// TIA Portal V21 export
// export: Created 2026-07-12T08:36:11.2898125Z, ExportSetting None, DisplayName Totally Integrated Automation Portal, DisplayVersion V21, DisplayName SINAMICS Startdrive Advanced, DisplayVersion V21, DisplayName SINAMICS Startdrive G110M, G120, G120C, G120D, G120P, G115D, DisplayVersion V21, DisplayName SINAMICS Startdrive G130, G150, S120, S150, G200, G220, S200, S210, S220, Innomotics MVD, DisplayVersion V21, DisplayName STEP 7 Professional, DisplayVersion V21, DisplayName STEP 7 Safety, DisplayVersion V21, DisplayName Tech WebApplication, DisplayVersion V21, DisplayName WinCC Basic/Comfort/Advanced, DisplayVersion V21, DisplayName WinCC Professional, DisplayVersion V21, DisplayName WinCC Unified, DisplayVersion V21
FUNCTION_BLOCK "FB_SingleSolCyl_SCL"   // FB2104, LAD
{ S7_Optimized_Access := 'TRUE' }
// stored: AutoNumber false, MemoryReserve 100, SetENOAutomatically false
   VAR_INPUT
      Enable : Bool := 1;   // 使能单控气缸控制块，FALSE时关闭输出并禁止动作
      Mode : Int;   // 模式选择：1=Manual手动，2=Auto自动；其它值报警
      Exe_Auto : Bool;   // 自动模式下的动作命令，1伸出，0缩回
      Exe_Manual : Bool;   // 手动模式下的动作命令，1伸出，0缩回
      Sensor_Ext : Bool;   // 气缸伸出到位检测信号
      Sensor_Home : Bool;   // 气缸缩回原点检测信号
      Reset : Bool;   // 报警复位命令，清除报警和报警代码
      Timeout : Time := T#3S;   // 伸出或缩回等待传感器到位的超时时间，例如T#5s
   END_VAR
   VAR_OUTPUT
      Q : Bool;   // 控制真实电磁阀Q点，TRUE气缸伸出，FALSE气缸缩回
      Error : Bool;   // 报警锁存输出，需要ResetAlarm清除
      Error_Status : Word;   // 报警代码：2模式无效，3传感器冲突，257伸出超时，258缩回超时
      Extend : Bool;   // 当前有效模式下的伸出命令
      Retract : Bool;   // 当前有效模式下的缩回命令
      AutoActive : Bool;   // 自动模式有效状态：Enable、Mode=2、无报警
      ManualActive : Bool;   // 手动模式有效状态：Enable、Mode=1、无报警
   END_VAR
   VAR
      ExtendTimeoutTimer : TON_TIME;   // 伸出动作超时TON实例
      RetractTimeoutTimer : TON_TIME;   // 缩回动作超时TON实例
   END_VAR
BEGIN

REGION Network 1 (SCL): 条件判断集中处理
   // 报警、动作命令、伸出/缩回超时集中在本SCL程序段处理；ManualActive、AutoActive和Q输出保留LAD程序段。
   // 条件集中处理：报警、命令、超时都放在本SCL程序段
   // 保留LAD程序段只负责：ManualActive、AutoActive、Q输出

   // Reset优先清除报警；若故障原因仍存在，后续逻辑会重新报警
   IF #Reset THEN
       #Error := FALSE;
       #Error_Status := W#16#0000;
   END_IF;

   // 默认先清除动作命令，避免无效模式或报警时误动作
   #Extend := FALSE;
   #Retract := FALSE;

   // 根据有效模式生成动作命令：1伸出，0缩回
   IF #Enable AND NOT #Error THEN
       IF #ManualActive THEN
           #Extend := #Exe_Manual;
           #Retract := NOT #Exe_Manual;
       ELSIF #AutoActive THEN
           #Extend := #Exe_Auto;
           #Retract := NOT #Exe_Auto;
       END_IF;
   END_IF;

   // 定时器集中调用：伸出等待Sensor_Ext，缩回等待Sensor_Home
   #ExtendTimeoutTimer(IN := #Extend AND NOT #Sensor_Ext,
                       PT := #Timeout);
   #RetractTimeoutTimer(IN := #Retract AND NOT #Sensor_Home,
                        PT := #Timeout);

   // 报警判断集中处理
   IF #Enable AND NOT #Error THEN
       // Mode只能为1或2；
       IF (#Mode <> 1) AND (#Mode <> 2) THEN
           #Error := TRUE;
           #Error_Status := W#16#0002;

       // 两个极限传感器不能同时为1
       ELSIF #Sensor_Ext AND #Sensor_Home THEN
           #Error := TRUE;
           #Error_Status := W#16#0003;

       // 伸出不到位超时
       ELSIF #ExtendTimeoutTimer.Q THEN
           #Error := TRUE;
           #Error_Status := W#16#0101;

       // 缩回不到位超时
       ELSIF #RetractTimeoutTimer.Q THEN
           #Error := TRUE;
           #Error_Status := W#16#0102;
       END_IF;
   END_IF;

   // 报警后本扫描周期立即撤销有效模式和动作命令，后续LAD Q输出保持安全关闭
   IF #Error THEN
       #ManualActive := FALSE;
       #AutoActive := FALSE;
       #Extend := FALSE;
       #Retract := FALSE;
   END_IF;
END_REGION

REGION Network 2: Manual模式有效
   // Mode=1时手动模式有效，只允许ManualCmd控制气缸。
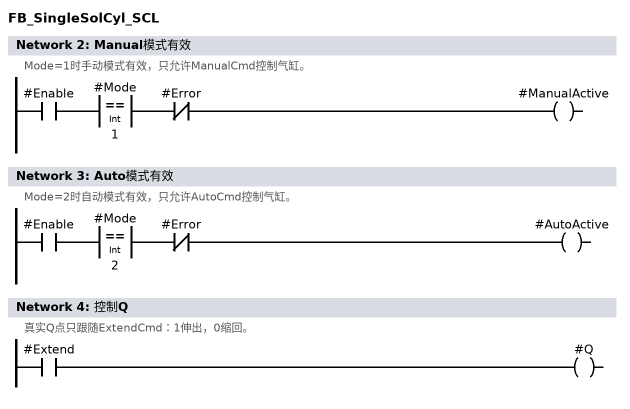
   RUNG wire#powerrail
      Contact( #Enable )
      { S7_Templates := "SrcType := Int" } EQ_Contact(in1 := #Mode, in2 := 1)
      I_Contact( #Error )
      Coil( #ManualActive )
   END_RUNG
   // the same network as SCL:
   #ManualActive := #Enable AND (#Mode = 1) AND NOT #Error;
END_REGION

REGION Network 3: Auto模式有效
   // Mode=2时自动模式有效，只允许AutoCmd控制气缸。
   RUNG wire#powerrail
      Contact( #Enable )
      { S7_Templates := "SrcType := Int" } EQ_Contact(in1 := #Mode, in2 := 2)
      I_Contact( #Error )
      Coil( #AutoActive )
   END_RUNG
   // the same network as SCL:
   #AutoActive := #Enable AND (#Mode = 2) AND NOT #Error;
END_REGION

REGION Network 4: 控制Q
   // 真实Q点只跟随ExtendCmd：1伸出，0缩回。
   RUNG wire#powerrail
      Contact( #Extend )
      Coil( #Q )
   END_RUNG
   // the same network as SCL:
   #Q := #Extend;
END_REGION
END_FUNCTION_BLOCK
